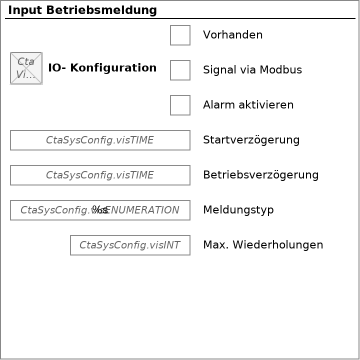
VISUALIZATION VIS_ANTRIEB_PARAMETER_IO1  // 360x360
VAR_INPUT
    ITF_ANTRIEBIN   :   ITF_ANTRIEB;
	ITF_IsOn_IN		:	CtaSysIO.ITF_IO;	
END_VAR
    Label (5,0 350x20), "Input Betriebsmeldung"
    Frame (170,25 20x20)
        shows CtaSysConfig.visBOOL(visfbBOOLIn := ITF_ANTRIEBIN.P_scIO_IsOn_fbxEnable)
    Label (200,25 150x20), "Vorhanden"
    Frame (170,60 20x20)
        shows CtaSysConfig.visBOOL(visfbBOOLIn := ITF_ANTRIEBIN.P_scIO_IsOn_fbxInputMb)
    Label (200,60 150x20), "Signal via Modbus"
    Frame (170,95 20x20)
        shows CtaSysConfig.visBOOL(visfbBOOLIn := ITF_ANTRIEBIN.P_scIO_IsOn_fbxDoesAlarm)
    Label (200,95 150x20), "Alarm aktivieren"
    Frame (10,130 180x20)
        shows CtaSysConfig.visTIME(visfbTIMEIn := ITF_ANTRIEBIN.P_scIO_IsOn_fbtDelayStart)
    Label (200,130 150x20), "Startverzögerung"
    Label (200,165 150x20), "Betriebsverzögerung"
    Frame (10,165 180x20)
        shows CtaSysConfig.visTIME(visfbTIMEIn := ITF_ANTRIEBIN.P_scIO_IsOn_fbtDelayRun)
    Frame (10,200 180x20)
        shows CtaSysConfig.visENUMERATION(visfbENUIn := ITF_ANTRIEBIN.P_scIO_IsOn_fbiTypeOfAck)
    Label (200,200 150x20), "Meldungstyp"
    Label (200,235 150x20), "Max. Wiederholungen"
    Line (5,18) (355,18)
    Frame (70,235 120x20)
        shows CtaSysConfig.visINT(visfbINTIn := ITF_ANTRIEBIN.P_scIO_IsOn_fbiMaxErrorRetryAllowed)
    Image (10,52 32x32), invisible if: ITF_IsOn_IN = 0, image: CtaVisSymbols.ImagePool.build
        OnMouseClick:  Dialog=VIS_ANTRIEB_POPUP_IO_ITF, Parameters={ITF_IO_IN: ITF_IsOn_IN}, OpenModal=True, OpenCentered=True
    Label (45,58 120x20), "IO- Konfiguration", invisible if: ITF_IsOn_IN = 0
    Textfield (30,200 140x20), "%s", text list: 'CtaAppReport.txtLibAp99_2enTypeOfAck', text index: CtaSysConfig.fcGetEnumerationId(ITF_ANTRIEBIN.P_scIO_IsOn_fbiTypeOfAck)
END_VISUALIZATION

// 40 Visualizations/POPUP/PARAMETER/AT_IO/VIS_ANTRIEB_PARAMETER_IO
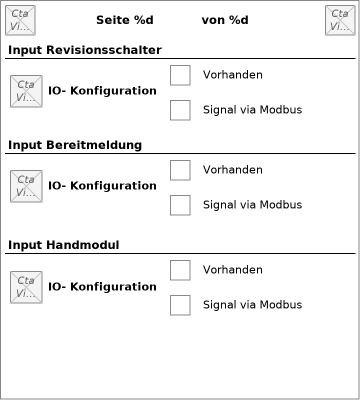
VISUALIZATION VIS_ANTRIEB_PARAMETER_IO  // 360x400
VAR_INPUT
    ITF_ANTRIEBIN    :   ITF_ANTRIEB;	
END_VAR
VAR
    uiPage  :   UINT;
    uiMin   :   UINT    := 0;
    uiMax   :   UINT    := 4;
END_VAR
    Frame (0,40 360x360), frame switch variable: uiPage
        shows VIS_ANTRIEB_PARAMETER_IO0(ITF_ANTRIEBIN := ITF_ANTRIEBIN, ITF_RevSwitch_IN := ITF_ANTRIEBIN.proRevisionSwitch_ITF, ITF_Ready_IN := ITF_ANTRIEBIN.proReady_ITF, ITF_HandModul_IN := ITF_ANTRIEBIN.proHandModul_ITF)
        shows VIS_ANTRIEB_PARAMETER_IO1(ITF_ANTRIEBIN := ITF_ANTRIEBIN, ITF_IsOn_IN := ITF_ANTRIEBIN.proIsOn_ITF)
        shows VIS_ANTRIEB_PARAMETER_IO2(ITF_ANTRIEBIN := ITF_ANTRIEBIN, ITF_NoError_IN := ITF_ANTRIEBIN.proNoError_ITF)
        shows VIS_ANTRIEB_PARAMETER_IO3(ITF_ANTRIEBIN := ITF_ANTRIEBIN, ITF_ActValue_IN := ITF_ANTRIEBIN.proActualValue_ITF)
        shows VIS_ANTRIEB_PARAMETER_IO4(ITF_ANTRIEBIN := ITF_ANTRIEBIN, ITF_xOn_IN := ITF_ANTRIEBIN.proOn_ITF, ITF_rOnY_IN := ITF_ANTRIEBIN.proOnY_ITF)
    Image (325,5 30x30), invisible if: uiPage = uiMax, image: CtaVisSymbols.ImagePool.arrow-right_square
        OnMouseClick: execute {
            uiPage := uiPage + 1;
            IF uiPage >= uiMax THEN
                uiPage := uiMax;
            END_IF;
        }
    Image (5,5 30x30), invisible if: uiPage = uiMin, image: CtaVisSymbols.ImagePool.arrow-left_square
        OnMouseClick: execute {
            uiPage := uiPage - 1;
            IF uiPage <= uiMin THEN
                uiPage := uiMin;
            END_IF;
        }
    Textfield (175,5 100x30), "von %d", text variable: uiMax
    Textfield (75,5 100x30), "Seite %d", text variable: uiPage
END_VISUALIZATION

// 40 Visualizations/POPUP/PARAMETER/AT_IO/VIS_ANTRIEB_PARAMETER_IO2
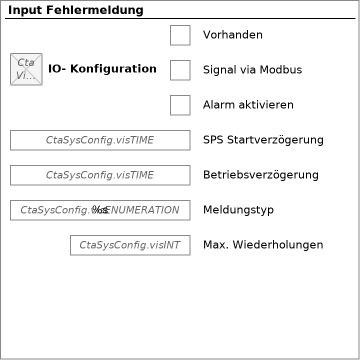
VISUALIZATION VIS_ANTRIEB_PARAMETER_IO2  // 360x360
VAR_INPUT
    ITF_ANTRIEBIN   :   ITF_ANTRIEB;
	ITF_NoError_IN	:	CtaSysIO.ITF_IO;	
END_VAR
    Label (5,0 350x20), "Input Fehlermeldung"
    Frame (170,25 20x20)
        shows CtaSysConfig.visBOOL(visfbBOOLIn := ITF_ANTRIEBIN.P_scIO_IsNoError_fbxEnable)
    Label (200,25 150x20), "Vorhanden"
    Frame (170,60 20x20)
        shows CtaSysConfig.visBOOL(visfbBOOLIn := ITF_ANTRIEBIN.P_scIO_IsNoError_fbxInputMb)
    Label (200,60 150x20), "Signal via Modbus"
    Frame (170,95 20x20)
        shows CtaSysConfig.visBOOL(visfbBOOLIn := ITF_ANTRIEBIN.P_scIO_IsNoError_fbxDoesAlarm)
    Label (200,95 150x20), "Alarm aktivieren"
    Frame (10,130 180x20)
        shows CtaSysConfig.visTIME(visfbTIMEIn := ITF_ANTRIEBIN.P_scIO_IsNoError_fbtDelayStartSps)
    Label (200,130 150x20), "SPS Startverzögerung"
    Label (200,165 150x20), "Betriebsverzögerung"
    Frame (10,165 180x20)
        shows CtaSysConfig.visTIME(visfbTIMEIn := ITF_ANTRIEBIN.P_scIO_IsNoError_fbtDelayRun)
    Frame (10,200 180x20)
        shows CtaSysConfig.visENUMERATION(visfbENUIn := ITF_ANTRIEBIN.P_scIO_IsNoError_fbiTypeOfAck)
    Label (200,200 150x20), "Meldungstyp"
    Label (200,235 150x20), "Max. Wiederholungen"
    Line (5,18) (355,18)
    Frame (70,235 120x20)
        shows CtaSysConfig.visINT(visfbINTIn := ITF_ANTRIEBIN.P_scIO_IsNoError_fbiMaxErrorRetryAllowed)
    Image (10,53 32x32), invisible if: ITF_NoError_IN = 0, image: CtaVisSymbols.ImagePool.build
        OnMouseClick:  Dialog=VIS_ANTRIEB_POPUP_IO_ITF, Parameters={ITF_IO_IN: ITF_NoError_IN}, OpenModal=True, OpenCentered=True
    Label (45,59 120x20), "IO- Konfiguration", invisible if: ITF_NoError_IN = 0
    Textfield (30,200 140x20), "%s", text list: 'CtaAppReport.txtLibAp99_2enTypeOfAck', text index: CtaSysConfig.fcGetEnumerationId(ITF_ANTRIEBIN.P_scIO_IsNoError_fbiTypeOfAck)
END_VISUALIZATION

// 40 Visualizations/POPUP/PARAMETER/AT_IO/VIS_ANTRIEB_PARAMETER_IO3
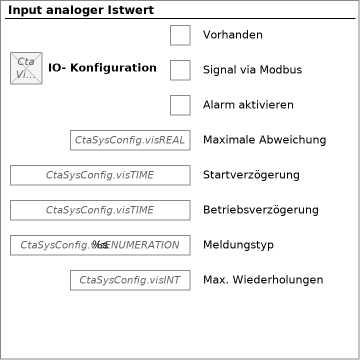
VISUALIZATION VIS_ANTRIEB_PARAMETER_IO3  // 360x360
VAR_INPUT
    ITF_ANTRIEBIN   	:   ITF_ANTRIEB;	
	ITF_ActValue_IN		:	CtaSysIO.ITF_IO;
END_VAR
    Label (5,0 350x20), "Input analoger Istwert"
    Frame (170,25 20x20)
        shows CtaSysConfig.visBOOL(visfbBOOLIn := ITF_ANTRIEBIN.P_scIO_IsValue_fbxEnable)
    Label (200,25 150x20), "Vorhanden"
    Frame (170,60 20x20)
        shows CtaSysConfig.visBOOL(visfbBOOLIn := ITF_ANTRIEBIN.P_scIO_IsValue_fbxInputMb)
    Label (200,60 150x20), "Signal via Modbus"
    Frame (170,95 20x20)
        shows CtaSysConfig.visBOOL(visfbBOOLIn := ITF_ANTRIEBIN.P_scIO_IsValue_fbxDoesAlarm)
    Label (200,95 150x20), "Alarm aktivieren"
    Frame (10,165 180x20)
        shows CtaSysConfig.visTIME(visfbTIMEIn := ITF_ANTRIEBIN.P_scIO_IsValue_fbtDelayStart)
    Label (200,165 150x20), "Startverzögerung"
    Label (200,200 150x20), "Betriebsverzögerung"
    Frame (10,200 180x20)
        shows CtaSysConfig.visTIME(visfbTIMEIn := ITF_ANTRIEBIN.P_scIO_IsValue_fbtDelayRun)
    Frame (70,130 120x20)
        shows CtaSysConfig.visREAL(visfbREALIn := ITF_ANTRIEBIN.P_scIO_IsValue_fbrMaxDiff, stPhysikalischeEinheit := '%')
    Label (200,130 150x20), "Maximale Abweichung"
    Label (200,235 150x20), "Meldungstyp"
    Label (200,270 150x20), "Max. Wiederholungen"
    Line (5,18) (355,18)
    Frame (10,235 180x20)
        shows CtaSysConfig.visENUMERATION(visfbENUIn := ITF_ANTRIEBIN.P_scIO_IsValue_fbiTypeOfAck)
    Frame (70,270 120x20)
        shows CtaSysConfig.visINT(visfbINTIn := ITF_ANTRIEBIN.P_scIO_IsValue_fbiMaxErrorRetryAllowed)
    Image (10,52 32x32), invisible if: ITF_ActValue_IN = 0, image: CtaVisSymbols.ImagePool.build
        OnMouseClick:  Dialog=VIS_ANTRIEB_POPUP_IO_ITF, Parameters={ITF_IO_IN: ITF_ActValue_IN}, OpenModal=True, OpenCentered=True
    Label (45,58 120x20), "IO- Konfiguration", invisible if: ITF_ActValue_IN = 0
    Textfield (30,235 140x20), "%s", text list: 'CtaAppReport.txtLibAp99_2enTypeOfAck', text index: CtaSysConfig.fcGetEnumerationId(ITF_ANTRIEBIN.P_scIO_IsValue_fbiTypeOfAck)
END_VISUALIZATION

// 40 Visualizations/POPUP/PARAMETER/AT_InfluxDb/VIS_ANTRIEB_PARAMETER_TRENDLOG
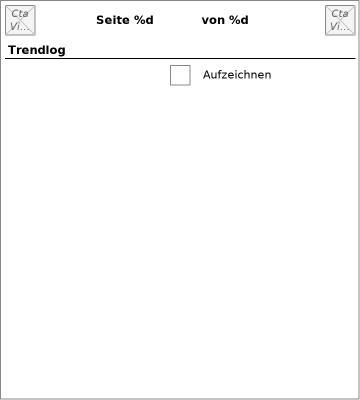
VISUALIZATION VIS_ANTRIEB_PARAMETER_TRENDLOG  // 360x400
VAR_INPUT
    ITF_ANTRIEBIN    :   ITF_ANTRIEB;	
END_VAR
VAR
    uiPage  :   UINT;
    uiMin   :   UINT    := 0;
    uiMax   :   UINT    := 0;
END_VAR
    Image (5,5 30x30), invisible if: uiPage = uiMin, image: CtaVisSymbols.ImagePool.arrow-left_square
        OnMouseClick: execute {
            uiPage := uiPage - 1;
            IF uiPage <= uiMin THEN
                uiPage := uiMin;
            END_IF;
        }
    Image (325,5 30x30), invisible if: uiPage = uiMax, image: CtaVisSymbols.ImagePool.arrow-right_square
        OnMouseClick: execute {
            uiPage := uiPage + 1;
            IF uiPage >= uiMax THEN
                uiPage := uiMax;
            END_IF;
        }
    Frame (0,40 360x360), frame switch variable: uiPage
        shows VIS_ANTRIEB_PARAMETER_TRENDLOG0(ITF_ANTRIEBIN := ITF_ANTRIEBIN)
        shows AT_ParameterIO1(ITF_Parameter := ITF_Parameter)
        pReferences[0]: ITF_Parameter=ITF_Parameter
    Textfield (75,5 100x30), "Seite %d", text variable: uiPage
    Textfield (175,5 100x30), "von %d", text variable: uiMax
END_VISUALIZATION

// 40 Visualizations/POPUP/PARAMETER/AT_InfluxDb/VIS_ANTRIEB_PARAMETER_TRENDLOG0
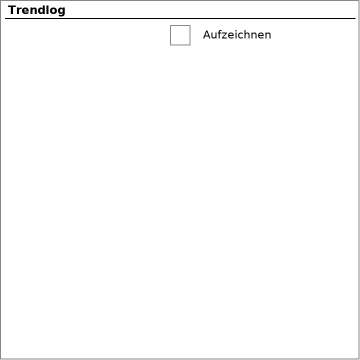
VISUALIZATION VIS_ANTRIEB_PARAMETER_TRENDLOG0  // 360x360
VAR_INPUT
    ITF_ANTRIEBIN    :   ITF_ANTRIEB;	
END_VAR
    Frame (170,25 20x20)
        shows CtaSysConfig.visBOOL(visfbBOOLIn := ITF_ANTRIEBIN.P_scInfluxDb_fbxEnable)
    Label (200,25 150x20), "Aufzeichnen"
    Label (5,0 350x20), "Trendlog"
    Line (5,18) (355,18)
END_VISUALIZATION

// 40 Visualizations/POPUP/IO/VIS_ANTRIEB_IO0
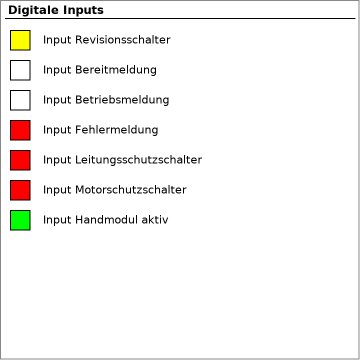
VISUALIZATION VIS_ANTRIEB_IO0  // 360x360
VAR_INPUT
    ITF_ANTRIEBIN    :   ITF_ANTRIEB;	
END_VAR
    Label (40,30 320x20), "Input Revisionsschalter", invisible if: ITF_ANTRIEBIN.proNotShowDI_RevisionSwitchOk
    Label (40,60 320x20), "Input Bereitmeldung", invisible if: ITF_ANTRIEBIN.proNotShowDI_Ready
    Rectangle (10,30 20x20), colour toggle: ITF_ANTRIEBIN.proGetDI_RevisionSwitchOK, invisible if: ITF_ANTRIEBIN.proNotShowDI_RevisionSwitchOk
    Rectangle (10,60 20x20), colour toggle: ITF_ANTRIEBIN.proGetDI_IsReady, invisible if: ITF_ANTRIEBIN.proNotShowDI_Ready
    Label (40,120 320x20), "Input Fehlermeldung", invisible if: ITF_ANTRIEBIN.proNotShowDI_NoError
    Rectangle (10,120 20x20), colour toggle: ITF_ANTRIEBIN.proGetDI_NoError, invisible if: ITF_ANTRIEBIN.proNotShowDI_NoError
    Rectangle (10,150 20x20), colour toggle: ITF_ANTRIEBIN.proGetDI_FuseOK, invisible if: ITF_ANTRIEBIN.proNotShowDI_FuseOk
    Label (40,150 320x20), "Input Leitungsschutzschalter", invisible if: ITF_ANTRIEBIN.proNotShowDI_FuseOk
    Label (40,180 320x20), "Input Motorschutzschalter", invisible if: ITF_ANTRIEBIN.proNotShowDI_MotorFuseOk
    Rectangle (10,180 20x20), colour toggle: ITF_ANTRIEBIN.proGetDI_MotorFuseOk, invisible if: ITF_ANTRIEBIN.proNotShowDI_MotorFuseOk
    Label (40,210 320x20), "Input Handmodul aktiv", invisible if: ITF_ANTRIEBIN.proNotShowDI_MotorHand
    Rectangle (10,210 20x20), colour toggle: ITF_ANTRIEBIN.proGetDI_MotorHand, invisible if: ITF_ANTRIEBIN.proNotShowDI_MotorHand
    Label (40,90 320x20), "Input Betriebsmeldung", invisible if: ITF_ANTRIEBIN.proNotShowDI_IsOn
    Rectangle (10,90 20x20), colour toggle: ITF_ANTRIEBIN.proGetDI_IsOn, invisible if: ITF_ANTRIEBIN.proNotShowDI_IsOn
    Label (5,0 350x20), "Digitale Inputs"
    Line (5,18) (355,18)
END_VISUALIZATION

// 40 Visualizations/POPUP/IO/VIS_ANTRIEB_IO
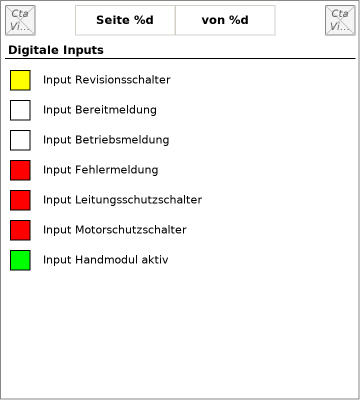
VISUALIZATION VIS_ANTRIEB_IO  // 360x400
VAR_INPUT
    ITF_ANTRIEBIN    :   ITF_ANTRIEB;	
END_VAR
VAR
    uiPage  :   UINT;
    uiMin   :   UINT    := 0;
    uiMax   :   UINT    := 1;
END_VAR
    Frame (0,40 360x360), frame switch variable: uiPage
        shows VIS_ANTRIEB_IO0(ITF_ANTRIEBIN := ITF_ANTRIEBIN)
        shows VIS_ANTRIEB_IO1(ITF_ANTRIEBIN := ITF_ANTRIEBIN)
        shows AT_ParameterIO2(ITF_Parameter := ITF_Parameter)
        shows AT_ParameterIO3(ITF_Parameter := ITF_Parameter)
    Image (325,5 30x30), invisible if: uiPage = uiMax, image: CtaVisSymbols.ImagePool.arrow-right_square
        OnMouseClick: execute {
            uiPage := uiPage + 1;
            IF uiPage >= uiMax THEN
                uiPage := uiMax;
            END_IF;
        }
    Image (5,5 30x30), invisible if: uiPage = uiMin, image: CtaVisSymbols.ImagePool.arrow-left_square
        OnMouseClick: execute {
            uiPage := uiPage - 1;
            IF uiPage <= uiMin THEN
                uiPage := uiMin;
            END_IF;
        }
    Textfield (175,5 100x30), "von %d", text variable: uiMax
    Textfield (75,5 100x30), "Seite %d", text variable: uiPage
END_VISUALIZATION

// 40 Visualizations/POPUP/IO/VIS_ANTRIEB_IO1
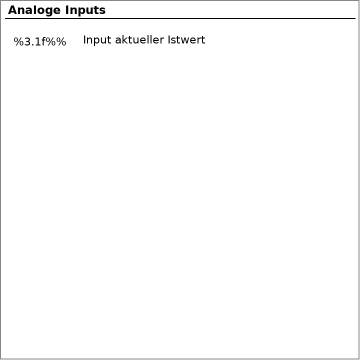
VISUALIZATION VIS_ANTRIEB_IO1  // 360x360
VAR_INPUT
    ITF_ANTRIEBIN    :   ITF_ANTRIEB;	
END_VAR
    Label (80,30 280x20), "Input aktueller Istwert", invisible if: ITF_ANTRIEBIN.proNotShowAI_ActualValue
    Label (5,0 350x20), "Analoge Inputs"
    Textfield (10,32 60x20), "%3.1f%%", text variable: ITF_ANTRIEBIN.proGetAI_ActualValue, invisible if: ITF_ANTRIEBIN.proNotShowAI_ActualValue
    Line (5,18) (355,18)
END_VISUALIZATION

// 40 Visualizations/ICON/ANTRIEB_BASE/ValueUpDwn
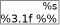
VISUALIZATION ValueUpDwn  // 60x25
VAR_INPUT
    ITF_ANTRIEB_IN   :   ITF_ANTRIEB;	
END_VAR
VAR_INPUT CONSTANT
    uiTextAusrichtung   : UINT := 4;    // 0 = Oben links | 1 = Horizontal zentriert | 2 = Rechts | 4 = Vertikal zentriert | 8 = Unten
END_VAR
    Textfield (0,0 60x12), "%s", text variable: ITF_ANTRIEB_IN.proGetBMK, invisible if: ITF_ANTRIEB_IN.proNoBmkInList
        p3718999670: uiTextAusrichtung
    Textfield (0,13 60x12), "%3.1f %%", text variable: ITF_ANTRIEB_IN.proOnY, invisible if: NOT ITF_ANTRIEB_IN.proIsRegulatet
        p3718999670: uiTextAusrichtung
END_VISUALIZATION

// 40 Visualizations/ICON/ANTRIEB_LEFT/ANTRIEB_LEFT_ABOVE/VIS_ANTRIEB_LEFT_ABOVE
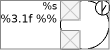
VISUALIZATION VIS_ANTRIEB_LEFT_ABOVE  // 110x50
VAR_INPUT
    ITF_ANTRIEB_IN   	:   ITF_ANTRIEB;
END_VAR
VAR_INPUT CONSTANT
	stExklParameter		:	STRING[40] := ' ';
END_VAR
VAR CONSTANT
	uiIconnr		:	UINT := 0;
END_VAR
    Frame (0,0 110x50), invisible if: NOT fcCheckQuerryAndIconReturn(_ITF_IN := ITF_ANTRIEB_IN, _uiIconNr_IN := uiIconNr)
        shows VIS_ANTRIEB_LeftAboveCheckQuerry(ITF_ANTRIEB_IN := ITF_ANTRIEB_IN, stExklParameter := stExklParameter)
END_VISUALIZATION

// 40 Visualizations/ICON/ANTRIEB_LEFT/ANTRIEB_LEFT_ABOVE/VIS_ANTRIEB_LeftAboveCheckIsEnabled
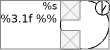
VISUALIZATION VIS_ANTRIEB_LeftAboveCheckIsEnabled  // 110x50
VAR_INPUT
    ITF_ANTRIEB_IN   :   ITF_ANTRIEB;	
END_VAR
VAR_INPUT
	stExklParameter		:	STRING[40];
END_VAR
    Frame (60,0 50x50), invisible if: NOT ITF_ANTRIEB_IN.proIsEnabled
        shows Icon_Left(ITF_ANTRIEB_IN := ITF_ANTRIEB_IN)
    Frame (0,0 60x25), invisible if: NOT ITF_ANTRIEB_IN.proIsEnabled
        shows ValueUpDwn(ITF_ANTRIEB_IN := ITF_ANTRIEB_IN, uiTextAusrichtung := 6)
    Frame (95,0 15x15), invisible if: NOT ITF_ANTRIEB_IN.proIsEnabled
        shows CommandOn(ITF_ANTRIEB_IN := ITF_ANTRIEB_IN)
    Rectangle (0,0 110x50)
        OnMouseClick:  Dialog=POPUP_ANTRIEB, Parameters={stExklParameter_IN: stExklParameter, ITF_ANTRIEBIN: ITF_ANTRIEB_IN, uiPopUpGruppe: 0}, OpenCentered=True
END_VISUALIZATION

// 40 Visualizations/ICON/ANTRIEB_LEFT/ANTRIEB_LEFT_ABOVE/VIS_ANTRIEB_LeftAboveCheckQuerry
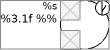
VISUALIZATION VIS_ANTRIEB_LeftAboveCheckQuerry  // 110x50
VAR_INPUT
    ITF_ANTRIEB_IN   :   ITF_ANTRIEB;	
END_VAR
VAR_INPUT
	stExklParameter		:	STRING[40];
END_VAR
    Frame (0,0 110x50)
        shows VIS_ANTRIEB_LeftAboveCheckIsEnabled(ITF_ANTRIEB_IN := ITF_ANTRIEB_IN, stExklParameter := stExklParameter)
END_VISUALIZATION

// 40 Visualizations/ICON/ANTRIEB_LEFT/ANTRIEB_LEFT_BELOW/VIS_ANTRIEB_LEFT_BELOW
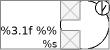
VISUALIZATION VIS_ANTRIEB_LEFT_BELOW  // 110x50
VAR_INPUT
    ITF_ANTRIEB_IN   :   ITF_ANTRIEB;	
END_VAR
VAR_INPUT
	stExklParameter		:	STRING[40] := ' ';
END_VAR
VAR CONSTANT
	uiIconNr		:	UINT := 1 ;
END_VAR
    Frame (0,0 110x50), invisible if: NOT fcCheckQuerryAndIconReturn(_ITF_IN := ITF_ANTRIEB_IN, _uiIconNr_IN := uiIconNr)
        shows VIS_ANTRIEB_LeftBelowCheckQuerry(ITF_ANTRIEB_IN := ITF_ANTRIEB_IN, stExklParameter := stExklParameter)
END_VISUALIZATION

// 40 Visualizations/ICON/ANTRIEB_LEFT/ANTRIEB_LEFT_BELOW/VIS_ANTRIEB_LeftBelowCheckIsEnabled
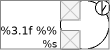
VISUALIZATION VIS_ANTRIEB_LeftBelowCheckIsEnabled  // 110x50
VAR_INPUT
    ITF_ANTRIEB_IN   :   ITF_ANTRIEB;	
END_VAR
VAR_INPUT
	stExklParameter		:	STRING[40];
END_VAR
    Frame (60,0 50x50), invisible if: NOT ITF_ANTRIEB_IN.proIsEnabled
        shows Icon_Left(ITF_ANTRIEB_IN := ITF_ANTRIEB_IN)
    Frame (0,25 60x27), invisible if: NOT ITF_ANTRIEB_IN.proIsEnabled
        shows ValueDwnUp(ITF_ANTRIEB_IN := ITF_ANTRIEB_IN, uiTextAusrichtung := 6)
    Frame (95,0 15x15), invisible if: NOT ITF_ANTRIEB_IN.proIsEnabled
        shows CommandOn(ITF_ANTRIEB_IN := ITF_ANTRIEB_IN)
    Rectangle (0,0 110x50)
        OnMouseClick:  Dialog=POPUP_ANTRIEB, Parameters={uiPopUpGruppe: 0, stExklParameter_IN: stExklParameter, ITF_ANTRIEBIN: ITF_ANTRIEB_IN}, OpenCentered=True
END_VISUALIZATION

// 40 Visualizations/ICON/ANTRIEB_LEFT/ANTRIEB_LEFT_BELOW/VIS_ANTRIEB_LeftBelowCheckQuerry
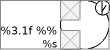
VISUALIZATION VIS_ANTRIEB_LeftBelowCheckQuerry  // 110x50
VAR_INPUT
    ITF_ANTRIEB_IN   :   ITF_ANTRIEB;	
END_VAR
VAR_INPUT
	stExklParameter		:	STRING[40];
END_VAR
    Frame (0,0 110x50)
        shows VIS_ANTRIEB_LeftBelowCheckIsEnabled(ITF_ANTRIEB_IN := ITF_ANTRIEB_IN, stExklParameter := stExklParameter)
END_VISUALIZATION

// 40 Visualizations/ICON/ANTRIEB_RIGHT/ANTRIEB_RIGHT_BELOW/VIS_ANTRIEB_RIGHT_BELOW
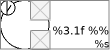
VISUALIZATION VIS_ANTRIEB_RIGHT_BELOW  // 110x50
VAR_INPUT
    ITF_ANTRIEB_IN   :   ITF_ANTRIEB;	
END_VAR
VAR_INPUT CONSTANT
	stExklParameter		:	STRING[40] := ' ';
END_VAR
VAR CONSTANT
	uiIconNr		:	UINT := 3;
END_VAR
    Frame (0,0 110x50), invisible if: NOT fcCheckQuerryAndIconReturn(_ITF_IN := ITF_ANTRIEB_IN, _uiIconNr_IN := uiIconNr)
        shows VIS_ANTRIEB_RigthBelowCheckQuerry(ITF_ANTRIEB_IN := ITF_ANTRIEB_IN, stExklParameter := stExklParameter)
END_VISUALIZATION

// 40 Visualizations/ICON/ANTRIEB_RIGHT/ANTRIEB_RIGHT_BELOW/VIS_ANTRIEB_RigthBelowCheckIsEnabled
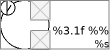
VISUALIZATION VIS_ANTRIEB_RigthBelowCheckIsEnabled  // 110x50
VAR_INPUT
    ITF_ANTRIEB_IN   :   ITF_ANTRIEB;	
END_VAR
VAR_INPUT
	stExklParameter		:	STRING[40];
END_VAR
    Frame (0,0 50x50), invisible if: NOT ITF_ANTRIEB_IN.proIsEnabled
        shows Icon_Right(ITF_ANTRIEB_IN := ITF_ANTRIEB_IN)
    Frame (52,25 60x27), invisible if: NOT ITF_ANTRIEB_IN.proIsEnabled
        shows ValueDwnUp(ITF_ANTRIEB_IN := ITF_ANTRIEB_IN, uiTextAusrichtung := 4)
    Frame (0,0 15x15), invisible if: NOT ITF_ANTRIEB_IN.proIsEnabled
        shows CommandOn(ITF_ANTRIEB_IN := ITF_ANTRIEB_IN)
    Rectangle (0,0 110x50)
        OnMouseClick:  Dialog=POPUP_ANTRIEB, Parameters={uiPopUpGruppe: 0, stExklParameter_IN: stExklParameter, ITF_ANTRIEBIN: ITF_ANTRIEB_IN}, OpenCentered=True
END_VISUALIZATION

// 40 Visualizations/ICON/ANTRIEB_RIGHT/ANTRIEB_RIGHT_BELOW/VIS_ANTRIEB_RigthBelowCheckQuerry
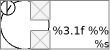
VISUALIZATION VIS_ANTRIEB_RigthBelowCheckQuerry  // 110x50
VAR_INPUT
    ITF_ANTRIEB_IN   :   ITF_ANTRIEB;	
END_VAR
VAR_INPUT
	stExklParameter		:	STRING[40];
END_VAR
    Frame (0,0 110x50)
        shows VIS_ANTRIEB_RigthBelowCheckIsEnabled(ITF_ANTRIEB_IN := ITF_ANTRIEB_IN, stExklParameter := stExklParameter)
END_VISUALIZATION

// 40 Visualizations/ICON/ANTRIEB_BASE/ICON/Icon_Right
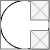
VISUALIZATION Icon_Right  // 50x50
VAR_INPUT
    ITF_ANTRIEB_IN   :   ITF_ANTRIEB;	
END_VAR
    Ellipse (0,0 49x49), colour toggle: ITF_ANTRIEB_IN.proMotorIsOn, invisible if: ITF_ANTRIEB_IN.proIsError
    Ellipse (0,0 49x49), colour toggle: ITF_ANTRIEB_IN.proIsError
    Image (30,0 20x20), invisible if: NOT ITF_ANTRIEB_IN.proIsWarning, image: CtaVisSymbols.ImagePool.CtaWarning
    Image (30,30 20x20), invisible if: NOT ITF_ANTRIEB_IN.proIsHandOnOrOff, image: CtaVisSymbols.ImagePool.front_hand_Yellow
    Image (30,30 20x20), invisible if: NOT ITF_ANTRIEB_IN.proHandOff, image: CtaVisSymbols.ImagePool.front_hand_Yellow_Off
END_VISUALIZATION

// 40 Visualizations/POPUP/PARAMETER/AT_IO/VIS_ANTRIEB_PARAMETER_IO4
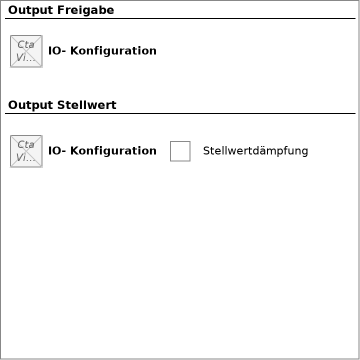
VISUALIZATION VIS_ANTRIEB_PARAMETER_IO4  // 360x360
VAR_INPUT
    ITF_ANTRIEBIN   :   ITF_ANTRIEB;	
	ITF_xOn_IN		:	CtaSysIO.ITF_IO;
	ITF_rOnY_IN		:	CtaSysIO.ITF_IO;
END_VAR
    Label (5,0 350x20), "Output Freigabe"
    Label (5,95 350x20), "Output Stellwert"
    Line (5,113) (355,113)
    Line (5,18) (355,18)
    Image (10,35 32x32), invisible if: ITF_xOn_IN = 0, image: CtaVisSymbols.ImagePool.build
        OnMouseClick:  Dialog=VIS_ANTRIEB_POPUP_IO_ITF, Parameters={ITF_IO_IN: ITF_xOn_IN}, OpenModal=True, OpenCentered=True
    Image (10,135 32x32), invisible if: ITF_rOnY_IN = 0, image: CtaVisSymbols.ImagePool.build
        OnMouseClick:  Dialog=VIS_ANTRIEB_POPUP_IO_ITF, Parameters={ITF_IO_IN: ITF_rOnY_IN}, OpenModal=True, OpenCentered=True
    Label (45,41 120x20), "IO- Konfiguration", invisible if: ITF_xOn_IN = 0
    Label (45,141 120x20), "IO- Konfiguration", invisible if: ITF_rOnY_IN = 0
    Label (200,141 150x20), "Stellwertdämpfung"
    Frame (170,141 20x20)
        shows CtaAppDumper.VisDumperSmall(fbDumper := ITF_ANTRIEBIN.proRefToRonYDumper)
END_VISUALIZATION

// 40 Visualizations/POPUP/PARAMETER/VIS_ANTRIEB_POPUP_IO_ITF
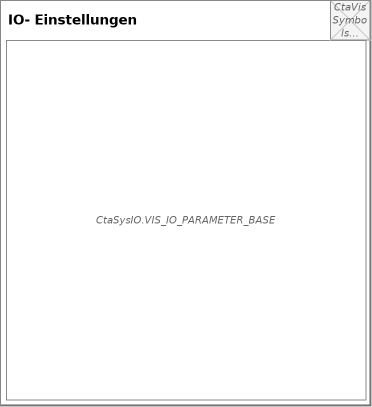
VISUALIZATION VIS_ANTRIEB_POPUP_IO_ITF  // 372x407
VAR_INPUT
    ITF_IO_IN    :   CtaSysIO.ITF_IO;	
END_VAR
    RoundedRectangle (0,0 370x405)
    Frame (6,40 360x360)
        shows CtaSysIO.VIS_IO_PARAMETER_BASE(ITF_IO_IN := ITF_IO_IN)
        shows VIS_ANTRIEB_PARAMETER_IO1(ITF_ANTRIEBIN := ITF_ANTRIEBIN)
        shows VIS_ANTRIEB_PARAMETER_IO2(ITF_ANTRIEBIN := ITF_ANTRIEBIN)
        shows VIS_ANTRIEB_PARAMETER_IO3(ITF_ANTRIEBIN := ITF_ANTRIEBIN)
    Image (330,0 40x40), image: CtaVisSymbols.ImagePool.close_solo_black
        OnMouseClick:  Dialog=VIS_ANTRIEB_POPUP_IO_ITF, Result=None, NumpadKeypadSet=True
    Label (5,0 150x40), "IO- Einstellungen"
END_VISUALIZATION

// 40 Visualizations/ICON/ANTRIEB_BASE/ValueDwnUp
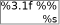
VISUALIZATION ValueDwnUp  // 60x25
VAR_INPUT
    ITF_ANTRIEB_IN   :   ITF_ANTRIEB;	
END_VAR
VAR_INPUT CONSTANT
    uiTextAusrichtung   : UINT := 4;    // 0 = Oben links | 1 = Horizontal zentriert | 2 = Rechts | 4 = Vertikal zentriert | 8 = Unten
END_VAR
    Textfield (0,0 60x12), "%3.1f %%", text variable: ITF_ANTRIEB_IN.proOnY, invisible if: NOT ITF_ANTRIEB_IN.proIsRegulatet
        p3718999670: uiTextAusrichtung
    Textfield (0,13 60x12), "%s", text variable: ITF_ANTRIEB_IN.proGetBMK, invisible if: ITF_ANTRIEB_IN.proNoBmkInList
        p3718999670: uiTextAusrichtung
END_VISUALIZATION

(* text list Error (id | default | de | en | fr | it)
  0 | keine Meldung Anstehend | Keine Meldung Anstehend | No message pending | Aucun message en attente | Nessun messaggio in sospeso
  1 | keine Betriebsrückmeldung | Keine Betriebsrückmeldung | No operational feedback | Aucune rétroaction opérationnelle | Nessun feedback operativo
  2 | Alarmkontakt Anstehend | Alarmkontakt Anstehend | Error contact pending | Contact d'alarme en attente | Contatto di allarme in sospeso
  3 | Leitungsschutzschalter ausfall | Leitungsschutzschalter ausfall | Circuit breaker failure | Défaillance du disjoncteur | Guasto dell'interruttore
  4 | Motorschutzschalter ausfall | Motorschutzschalter ausfall | Motor protection switch failure | Défaillance de l'interrupteur de protection du moteur | Guasto al salvamotore
  5 | Konfigurationsfehler speichern fehlgeschlagen reboot | Konfigurationsfehler speichern fehlgeschlagen reboot | Failed to save configuration error reboot | Impossible d'enregistrer l'erreur de configuration reboot | Impossibile salvare l'errore di configurazione reboot
   |  |  |  |  |  *)

(* text list Info (id | default | de | en | fr | it)
  0 | keine Meldung Anstehend | keine Meldung Anstehend | no message pending | aucun message en attente | nessun messaggio in sospeso
   |  |  |  |  |  *)

(* text list Warnung (id | default | de | en | fr | it)
  0 | Keine Meldung Anstehend | Keine Meldung Anstehend | No message pending | Aucun message en attente | Nessun messaggio in sospeso
  4 | Wahlschalter Hand, Ein | Wahlschalter Hand, Ein | Selector switch hand on | Commutateur de sélection a main, Allumé | Selettore a mano, acceso
  3 | Wahlschalter Hand, Aus | Wahlschalter Hand, Aus | Selector switch hand off | Commutateur de sélection a main, Éteint | Selettore a mano, spento
  2 | Revisionsschalter Ausgeschalten | Revisionsschalter Ausgeschalten | Revision switch off | Commutateur révision Désactiver | Interruttore di revisione disattivato
  1 | Sicherheits Stopp | Sicherheits Stopp | Safety stop | Arrêt de sécurité | Sosta di sicurezza
  5 | Handmodul aktiv | Handmodul aktiv | Hand module active | Module manuel actif | Modulo manuale attivo
   |  |  |  |  |  *)
